(* PLC project Demo, ACME plc-programming plugin 1.0 *)
(* stored: creationDateTime 2026-01-01T00:00:00 *)

TYPE E_MotorState : (Idle, Running, Faulted);
END_TYPE

FUNCTION_BLOCK FB_Motor
  VAR_INPUT
    xStart : BOOL;
    xStop : BOOL;
    xFeedback : BOOL;
  END_VAR
  VAR_OUTPUT
    xRun : BOOL;
    xFault : BOOL;
  END_VAR
  VAR
    eState : E_MotorState;
    rtStart : R_TRIG;
    tonFeedback : TON;
  END_VAR

            rtStart(CLK := xStart);
tonFeedback(IN := (eState = E_MotorState#Running) AND NOT xFeedback, PT := T#3S);

CASE eState OF
    E_MotorState#Idle:
        IF rtStart.Q AND NOT xStop THEN
            eState := E_MotorState#Running;
        END_IF;
    E_MotorState#Running:
        IF xStop THEN
            eState := E_MotorState#Idle;
        ELSIF tonFeedback.Q THEN
            eState := E_MotorState#Faulted;
        END_IF;
    E_MotorState#Faulted:
        IF xStop THEN
            eState := E_MotorState#Idle;
        END_IF;
ELSE
    eState := E_MotorState#Idle;
END_CASE;

xRun := eState = E_MotorState#Running;
xFault := eState = E_MotorState#Faulted;
          
END_FUNCTION_BLOCK

PROGRAM Main
  VAR
    fbConveyor : FB_Motor;
  END_VAR

            fbConveyor(xStart := FALSE, xStop := FALSE, xFeedback := FALSE);
          
END_PROGRAM

CONFIGURATION Config
  RESOURCE Res ON PLC
    TASK MainTask(INTERVAL := T#10ms, PRIORITY := 1);
    PROGRAM MainInstance WITH MainTask : Main;
  END_RESOURCE
END_CONFIGURATION
